// Mitsubishi GX Works2 project: 逆物料方向顺序启动   PLC: FX1S

PROGRAM MAIN
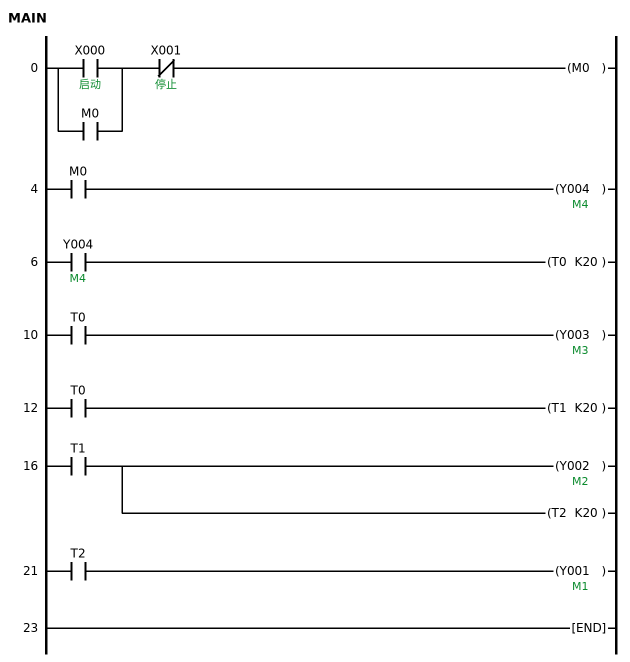
0     LD      X000  ; 启动
      OR      M0
      ANI     X001  ; 停止
      OUT     M0
4     LD      M0
      OUT     Y004  ; M4
6     LD      Y004  ; M4
      OUT     T0 K20
10    LD      T0
      OUT     Y003  ; M3
12    LD      T0
      OUT     T1 K20
16    LD      T1
      OUT     Y002  ; M2
      OUT     T2 K20
21    LD      T2
      OUT     Y001  ; M1
23    END
END_PROGRAM
